{attribute addProperty BoxType "EL3681-0000-0020"}
{attribute addProperty Id "SAI_InputsAT %I*SAI_Inputs_166EE3574860SAI_RangeAT %I*SAI_Range_DF9848341620SAI_Range_1AT %Q*SAI_Range_80D0ED7D1620WcStateAT %I*WcState_F855686C1620InfoDataAT %I*InfoData_BC63D37F80100"}
{attribute addProperty CRC "3586693794"}
{attribute addProperty SizeInBites "176"}
{attribute addProperty SizeInBytes "22"}
TYPE EL3681_AEC42720 :
STRUCT
	{attribute addProperty Name "SAI_Inputs"}
	SAI_Inputs : SAI_Inputs_166EE357;
	{attribute addProperty Name "SAI_Range"}
	SAI_Range : SAI_Range_DF984834;
	{attribute addProperty Name "SAI_Range_1"}
	SAI_Range_1 : SAI_Range_80D0ED7D;
	{attribute addProperty Name "WcState"}
	WcState : WcState_F855686C;
	{attribute addProperty Name "InfoData"}
	InfoData : InfoData_BC63D37F;
END_STRUCT
END_TYPE

(* stored: Version 1.2.0.0, ProductVersion 3.1.4024.9
   DUT EL3681_AEC42720: Id {511e34b3-5840-4885-95cb-3bd21426e76b} *)
